// TIA Portal V16 export
// export: Created 2023-09-25T11:31:52.9809725Z, ExportSetting WithDefaults, DisplayName Totally Integrated Automation Portal, DisplayVersion V16 Update 6, DisplayName TIA Portal Version Control Interface, DisplayVersion V16 Update 2, DisplayName TIA Portal Openness, DisplayVersion V16 Update 6, DisplayName STEP 7 Professional, DisplayVersion V16 Update 6, DisplayName STEP 7 Safety, DisplayVersion V16, DisplayName WinCC Advanced, DisplayVersion V16 Update 6
FUNCTION_BLOCK "06_M_Network connection control"   // FB10, LAD
TITLE = Sterowanie stycznikiem sieć
{ S7_Optimized_Access := 'TRUE' }
AUTHOR : rtecmer
VERSION : 0.1
// Sterowanie stycznikiem sieć. Ustawianie znaczników setCMD_SM i setSUPV_SM które przekazywane są do funkcji FC3/FC1 DRV01 driver napędów. Następnie przekazywane jest do warstwy Hardware/ OUT gdzie ustawiane jest wyjście sterownika
// stored: AutoNumber true, IsIECCheckEnabled false, IsRetainMemResEnabled false, MemoryReserve 500, SetENOAutomatically false, UDAEnableTagReadback false
   VAR_INPUT
      IsReady_M : Bool;   // Gotowość napędu
      IsModeAut : Bool;   // Znacznik tryb pracy
      Time_Off_Inverter : Bool;   // Bit Q - timer blokowania stycznika falownika po wyłączeniu
      setMotor2 : Bool;   // Znacznik dodatkowa pompy nr1
      setMotor3 : Bool;   // Znacznik ustawienie dodatkowej 2
      setMotor4 : Bool;   // Znacznik ustawienie dodatkowej 3
      IsRunNetwork_M : Bool;   // Potwierdzenie pracy z sieci M
      CMD_A_NetworkM : Bool;   // Znacznik serowania awaryjnego napędem z sieci w wypadku awarii falownika
   END_VAR
   VAR_IN_OUT
      TimerStartNetworkContactor : TON_TIME;   // Opóżnienie załaczenia stycznika sieć
      setCMD_SM : Bool;   // Znacznik sterowania stycznikiem sieć
      Is_extras_K1_M_1 : Bool;   // Znacznik motor dodatkowy nr 1
      Is_extras_K2_M_1 : Bool;   // Znacznik motor dodatkowy nr 2
      Is_extras_K3_M_1 : Bool;   // Znacznik motor dodatkowy nr 3
      setSUPV_SM : Bool;   // Znacznik polecenia sterowania z sieci
      off_add_K1 : Bool;   // znacznik pomocniczy podczas selektrywnego wyłączeania dodatkowej pompy
      off_add_K2 : Bool := false;   // znacznik pomocniczy podczas selektrywnego wyłączeania dodatkowej pompy
      off_add_K3 : Bool := false;   // znacznik pomocniczy podczas selektrywnego wyłączeania dodatkowej pompy
   END_VAR
   VAR
      tmpOFFinverter { ExternalAccessible := 'False'; ExternalVisible := 'False'; ExternalWritable := 'False'} : Bool;   // wyłączenie od osiągnięcia 50Hz + czas zwłoki
      mem_activ_K1 { ExternalAccessible := 'False'; ExternalVisible := 'False'; ExternalWritable := 'False'} : Bool;   // pamięć załączennie jako dodatkowa
      mem_activ_K2 { ExternalAccessible := 'False'; ExternalVisible := 'False'; ExternalWritable := 'False'} : Bool;   // pamięć załączennie jako dodatkowa
      mem_activ_K3 { ExternalAccessible := 'False'; ExternalVisible := 'False'; ExternalWritable := 'False'} : Bool;   // pamięć załączennie jako dodatkowa
   END_VAR
   VAR_TEMP   // added for the SCL form of the ladder/FBD networks
      _w1 : Bool;
   END_VAR
BEGIN

REGION Network 1: Timer opóźnienie dołączenie stycznika sieci
   // Histereza na dołączenie stycznika sieć po pracy z falownika
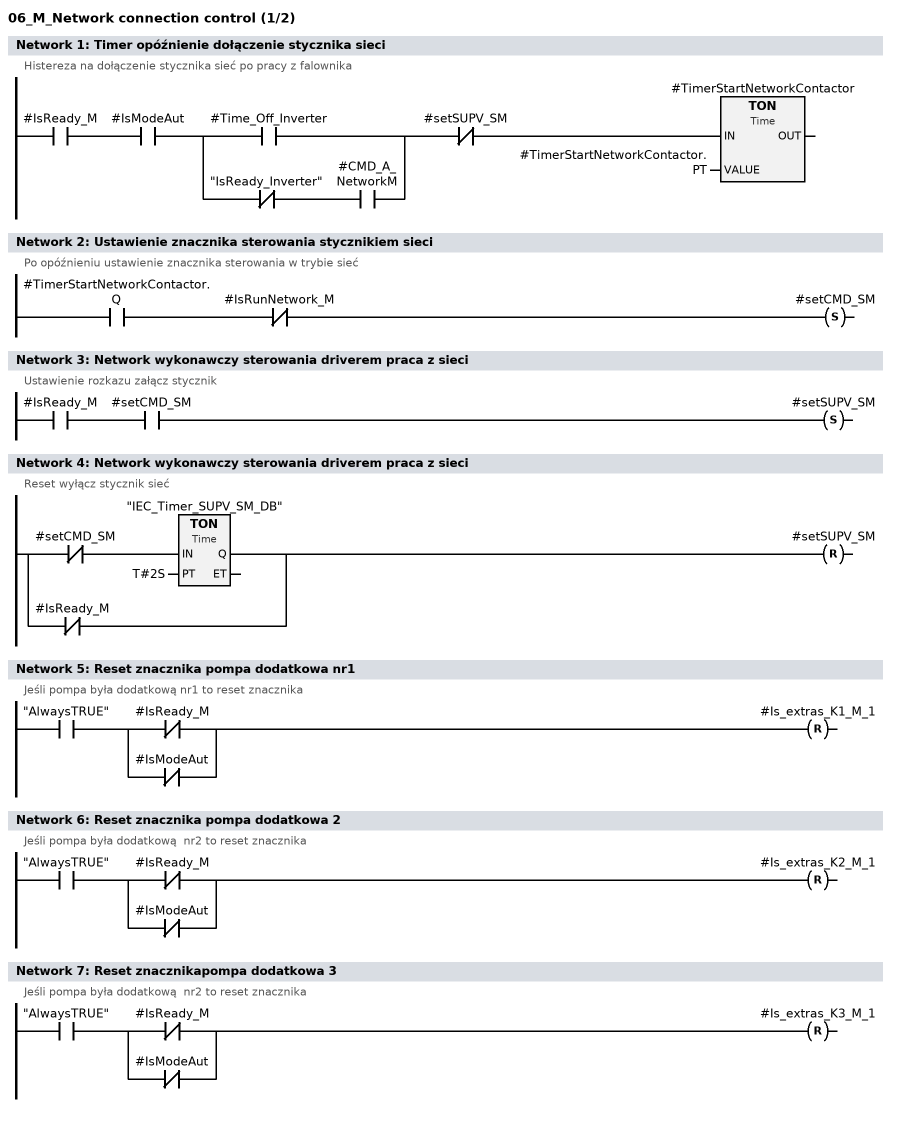
   #TimerStartNetworkContactor(IN := #IsReady_M AND #IsModeAut AND (#Time_Off_Inverter OR (NOT "IsReady_Inverter" AND #CMD_A_NetworkM)) AND NOT #setSUPV_SM, PT := #TimerStartNetworkContactor.PT);   // TON coil
END_REGION

REGION Network 2: Ustawienie znacznika sterowania stycznikiem sieci
   // Po opóźnieniu ustawienie znacznika sterowania w trybie sieć
   RUNG wire#powerrail
      Contact( #TimerStartNetworkContactor.Q )
      I_Contact( #IsRunNetwork_M )
      S_Coil( #setCMD_SM )
   END_RUNG
   // the same network as SCL:
   IF #TimerStartNetworkContactor.Q AND NOT #IsRunNetwork_M THEN #setCMD_SM := TRUE; END_IF;
END_REGION

REGION Network 3: Network wykonawczy sterowania driverem praca z sieci
   // Ustawienie rozkazu załącz stycznik
   RUNG wire#powerrail
      Contact( #IsReady_M )
      Contact( #setCMD_SM )
      S_Coil( #setSUPV_SM )
   END_RUNG
   // the same network as SCL:
   IF #IsReady_M AND #setCMD_SM THEN #setSUPV_SM := TRUE; END_IF;
END_REGION

REGION Network 4: Network wykonawczy sterowania driverem praca z sieci
   // Reset wyłącz stycznik sieć
   RUNG wire#powerrail
      I_Contact( #setCMD_SM )
      { S7_Templates := "time_type := Time" } "IEC_Timer_SUPV_SM_DB".TON(pt := T#2S, et =>)
      wire#w1
      R_Coil( #setSUPV_SM )
   END_RUNG
   RUNG wire#powerrail
      I_Contact( #IsReady_M )
   END_RUNG wire#w1
   // the same network as SCL:
   "IEC_Timer_SUPV_SM_DB".TON(IN := NOT #setCMD_SM, PT := T#2S);
   IF "IEC_Timer_SUPV_SM_DB".Q OR NOT #IsReady_M THEN #setSUPV_SM := FALSE; END_IF;
END_REGION

REGION Network 5: Reset znacznika pompa dodatkowa nr1
   // Jeśli pompa była dodatkową nr1 to reset znacznika
   RUNG wire#powerrail
      Contact( "AlwaysTRUE" )
      wire#w1
      I_Contact( #IsReady_M )
      wire#w2
      R_Coil( #Is_extras_K1_M_1 )
   END_RUNG
   RUNG wire#w1
      I_Contact( #IsModeAut )
   END_RUNG wire#w2
   // the same network as SCL:
   IF "AlwaysTRUE" AND (NOT #IsReady_M OR NOT #IsModeAut) THEN #Is_extras_K1_M_1 := FALSE; END_IF;
END_REGION

REGION Network 6: Reset znacznika pompa dodatkowa 2
   // Jeśli pompa była dodatkową  nr2 to reset znacznika
   RUNG wire#powerrail
      Contact( "AlwaysTRUE" )
      wire#w1
      I_Contact( #IsReady_M )
      wire#w2
      R_Coil( #Is_extras_K2_M_1 )
   END_RUNG
   RUNG wire#w1
      I_Contact( #IsModeAut )
   END_RUNG wire#w2
   // the same network as SCL:
   IF "AlwaysTRUE" AND (NOT #IsReady_M OR NOT #IsModeAut) THEN #Is_extras_K2_M_1 := FALSE; END_IF;
END_REGION

REGION Network 7: Reset znacznikapompa dodatkowa 3
   // Jeśli pompa była dodatkową  nr2 to reset znacznika
   RUNG wire#powerrail
      Contact( "AlwaysTRUE" )
      wire#w1
      I_Contact( #IsReady_M )
      wire#w2
      R_Coil( #Is_extras_K3_M_1 )
   END_RUNG
   RUNG wire#w1
      I_Contact( #IsModeAut )
   END_RUNG wire#w2
   // the same network as SCL:
   IF "AlwaysTRUE" AND (NOT #IsReady_M OR NOT #IsModeAut) THEN #Is_extras_K3_M_1 := FALSE; END_IF;
END_REGION

REGION Network 8: Reset Znacznika sterowania w trybie sieć
   // Gdy regulator PID ustawi szybkie wyłaczenie pompy dodatkowej nr 1, nr 2, nr 3 to następuje resetowania znacznika pracy pompy dodatkowej
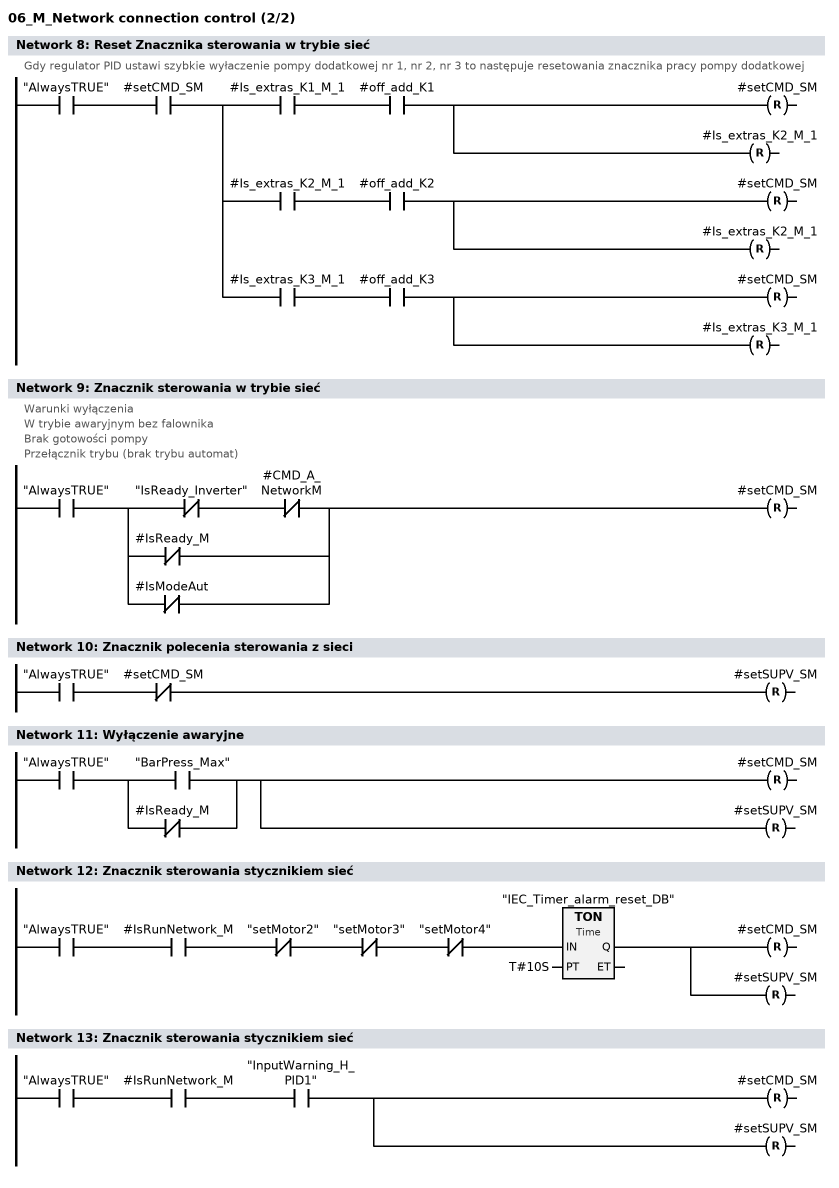
   RUNG wire#powerrail
      Contact( "AlwaysTRUE" )
      Contact( #setCMD_SM )
      wire#w1
      Contact( #Is_extras_K1_M_1 )
      Contact( #off_add_K1 )
      wire#w2
      R_Coil( #setCMD_SM )
   END_RUNG
   RUNG wire#w2
      R_Coil( #Is_extras_K2_M_1 )
   END_RUNG
   RUNG wire#w1
      Contact( #Is_extras_K2_M_1 )
      Contact( #off_add_K2 )
      wire#w3
      R_Coil( #setCMD_SM )
   END_RUNG
   RUNG wire#w3
      R_Coil( #Is_extras_K2_M_1 )
   END_RUNG
   RUNG wire#w1
      Contact( #Is_extras_K3_M_1 )
      Contact( #off_add_K3 )
      wire#w4
      R_Coil( #setCMD_SM )
   END_RUNG
   RUNG wire#w4
      R_Coil( #Is_extras_K3_M_1 )
   END_RUNG
   // the same network as SCL:
   #_w1 := "AlwaysTRUE" AND #setCMD_SM;
   IF #_w1 AND #Is_extras_K1_M_1 AND #off_add_K1 THEN
       #setCMD_SM := FALSE;
       #Is_extras_K2_M_1 := FALSE;
   END_IF;
   IF #_w1 AND #Is_extras_K2_M_1 AND #off_add_K2 THEN
       #setCMD_SM := FALSE;
       #Is_extras_K2_M_1 := FALSE;
   END_IF;
   IF #_w1 AND #Is_extras_K3_M_1 AND #off_add_K3 THEN
       #setCMD_SM := FALSE;
       #Is_extras_K3_M_1 := FALSE;
   END_IF;
END_REGION

REGION Network 9: Znacznik sterowania w trybie sieć
   // Warunki wyłączenia 
   // W trybie awaryjnym bez falownika
   // Brak gotowości pompy
   // Przełącznik trybu (brak trybu automat)
   RUNG wire#powerrail
      Contact( "AlwaysTRUE" )
      wire#w1
      I_Contact( "IsReady_Inverter" )
      I_Contact( #CMD_A_NetworkM )
      wire#w2
      R_Coil( #setCMD_SM )
   END_RUNG
   RUNG wire#w1
      I_Contact( #IsReady_M )
   END_RUNG wire#w2
   RUNG wire#w1
      I_Contact( #IsModeAut )
   END_RUNG wire#w2
   // the same network as SCL:
   IF "AlwaysTRUE" AND ((NOT "IsReady_Inverter" AND NOT #CMD_A_NetworkM) OR NOT #IsReady_M OR NOT #IsModeAut) THEN
       #setCMD_SM := FALSE;
   END_IF;
END_REGION

REGION Network 10: Znacznik polecenia sterowania z sieci
   RUNG wire#powerrail
      Contact( "AlwaysTRUE" )
      I_Contact( #setCMD_SM )
      R_Coil( #setSUPV_SM )
   END_RUNG
   // the same network as SCL:
   IF "AlwaysTRUE" AND NOT #setCMD_SM THEN #setSUPV_SM := FALSE; END_IF;
END_REGION

REGION Network 11: Wyłączenie awaryjne
   RUNG wire#powerrail
      Contact( "AlwaysTRUE" )
      wire#w1
      Contact( "BarPress_Max" )
      wire#w2
      R_Coil( #setCMD_SM )
   END_RUNG
   RUNG wire#w1
      I_Contact( #IsReady_M )
   END_RUNG wire#w2
   RUNG wire#w2
      R_Coil( #setSUPV_SM )
   END_RUNG
   // the same network as SCL:
   IF "AlwaysTRUE" AND ("BarPress_Max" OR NOT #IsReady_M) THEN
       #setCMD_SM := FALSE;
       #setSUPV_SM := FALSE;
   END_IF;
END_REGION

REGION Network 12: Znacznik sterowania stycznikiem sieć
   RUNG wire#powerrail
      Contact( "AlwaysTRUE" )
      Contact( #IsRunNetwork_M )
      I_Contact( "setMotor2" )
      I_Contact( "setMotor3" )
      I_Contact( "setMotor4" )
      { S7_Templates := "time_type := Time" } "IEC_Timer_alarm_reset_DB".TON(pt := T#10S, et =>)
      wire#w1
      R_Coil( #setCMD_SM )
   END_RUNG
   RUNG wire#w1
      R_Coil( #setSUPV_SM )
   END_RUNG
   // the same network as SCL:
   "IEC_Timer_alarm_reset_DB".TON(IN := "AlwaysTRUE" AND #IsRunNetwork_M AND NOT "setMotor2" AND NOT "setMotor3" AND NOT "setMotor4",
                           PT := T#10S);
   IF "IEC_Timer_alarm_reset_DB".Q THEN
       #setCMD_SM := FALSE;
       #setSUPV_SM := FALSE;
   END_IF;
END_REGION

REGION Network 13: Znacznik sterowania stycznikiem sieć
   RUNG wire#powerrail
      Contact( "AlwaysTRUE" )
      Contact( #IsRunNetwork_M )
      Contact( "InputWarning_H_PID1" )
      wire#w1
      R_Coil( #setCMD_SM )
   END_RUNG
   RUNG wire#w1
      R_Coil( #setSUPV_SM )
   END_RUNG
   // the same network as SCL:
   IF "AlwaysTRUE" AND #IsRunNetwork_M AND "InputWarning_H_PID1" THEN
       #setCMD_SM := FALSE;
       #setSUPV_SM := FALSE;
   END_IF;
END_REGION
END_FUNCTION_BLOCK
